TYPE ST_Message :
STRUCT
	eLogLevel:			E_LogLevel;
	nID:				UDINT;
	{attribute 'displaymode':='datetime'}
	nTimestamp:			ULINT;	
	sSource:			STRING(255);
	sMessage:			STRING(255);
	sDefault:			STRING(255);
	sArguments:			STRING(255);
	bActive:			BOOL;
END_STRUCT
END_TYPE

(* stored: Version 1.1.0.1
   DUT ST_Message: Id {3a6a707d-2fa5-4b7c-9941-24b715ac8048} *)
